(* LS Electric XG5000 project: counter_and_timer *)
(* PLC LSPLC *)

PROGRAM NewProgram (* task: Scan Program *)
VAR
    INST : CTU_DINT;
    INST1 : TON;
    off AT %IX0.0.2 : BOOL;
    on AT %IX0.0.1 : BOOL;
    onoff : BOOL;
    relay AT %QX0.0.1 : BOOL;
    relayoff : BOOL;
    sen1 AT %IX0.0.3 : BOOL;
    sen2 AT %IX0.0.4 : BOOL;
    START : BOOL;
    timeroff : BOOL;
END_VAR

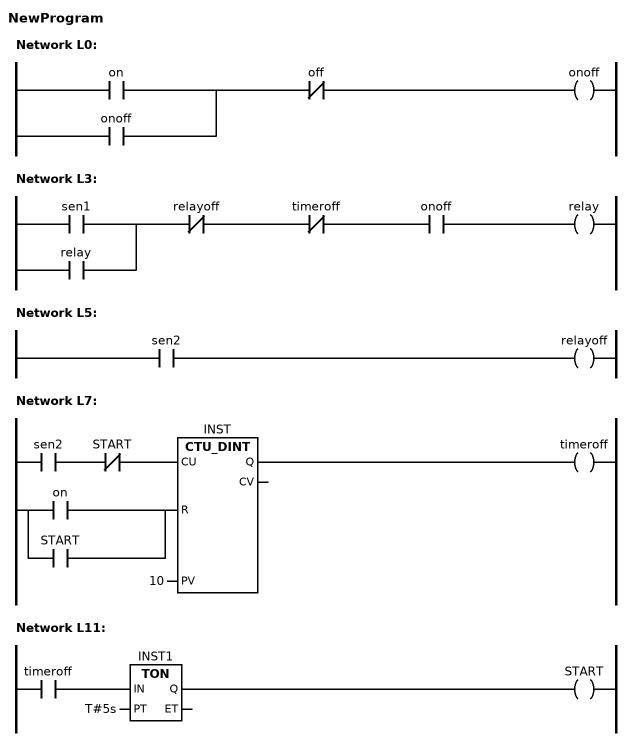
(* Rung L0 *)
onoff := (on OR onoff) AND NOT off;
(* Rung L3 *)
relay := (sen1 OR relay) AND NOT relayoff AND NOT timeroff AND onoff;
(* Rung L5 *)
relayoff := sen2;
(* Rung L7 *)
INST(CU := sen2 AND NOT START, R := on OR START, PV := 10);
timeroff := INST.Q;
(* Rung L11 *)
INST1(IN := timeroff, PT := T#5s);
START := INST1.Q;
END_PROGRAM